// TIA Portal V20 export
VAR_GLOBAL   // PLC tag table "im"
   "i0.0" AT %I0.0 : Bool;
   "i0.1" AT %I0.1 : Bool;
   "i0.2" AT %I0.2 : Bool;
   "i0.3" AT %I0.3 : Bool;
   "i0.4" AT %I0.4 : Bool;
   "i0.5" AT %I0.5 : Bool;
   "i0.6" AT %I0.6 : Bool;
   "i0.7" AT %I0.7 : Bool;
   "i1.0" AT %I1.0 : Bool;
   "i1.1" AT %I1.1 : Bool;
   "i1.2" AT %I1.2 : Bool;
   "i1.3" AT %I1.3 : Bool;
   "i1.4" AT %I1.4 : Bool;
   "i1.5" AT %I1.5 : Bool;
   "i1.6" AT %I1.6 : Bool;
   "i1.7" AT %I1.7 : Bool;
   "i2.0" AT %I2.0 : Bool;
   "i2.1" AT %I2.1 : Bool;
   "i2.2" AT %I2.2 : Bool;
   "i2.3" AT %I2.3 : Bool;
   "i2.4" AT %I2.4 : Bool;
   "i2.5" AT %I2.5 : Bool;
   "i2.6" AT %I2.6 : Bool;
   "i2.7" AT %I2.7 : Bool;
   "i3.0" AT %I3.0 : Bool;
   "i3.1" AT %I3.1 : Bool;
   "i3.2" AT %I3.2 : Bool;
   "i3.3" AT %I3.3 : Bool;
   "i3.4" AT %I3.4 : Bool;
   "i3.5" AT %I3.5 : Bool;
   "i3.6" AT %I3.6 : Bool;
   "i3.7" AT %I3.7 : Bool;
   "i4.0" AT %I4.0 : Bool;
   "i4.1" AT %I4.1 : Bool;
   "i4.2" AT %I4.2 : Bool;
   "i4.3" AT %I4.3 : Bool;
   "i4.4" AT %I4.4 : Bool;
   "i4.5" AT %I4.5 : Bool;
   "i4.6" AT %I4.6 : Bool;
   "i4.7" AT %I4.7 : Bool;
   "i5.0" AT %I5.0 : Bool;
   "i5.1" AT %I5.1 : Bool;
   "i5.2" AT %I5.2 : Bool;
   "i5.3" AT %I5.3 : Bool;
   "i5.4" AT %I5.4 : Bool;
   "i5.5" AT %I5.5 : Bool;
   "i5.6" AT %I5.6 : Bool;
   "i5.7" AT %I5.7 : Bool;
   "i6.0" AT %I6.0 : Bool;
   "i6.1" AT %I6.1 : Bool;
   "i6.2" AT %I6.2 : Bool;
   "i6.3" AT %I6.3 : Bool;
   "i6.4" AT %I6.4 : Bool;
   "i6.5" AT %I6.5 : Bool;
   "i6.6" AT %I6.6 : Bool;
   "i6.7" AT %I6.7 : Bool;
   "i7.0" AT %I7.0 : Bool;
   "i7.1" AT %I7.1 : Bool;
   "i7.2" AT %I7.2 : Bool;
   "i7.3" AT %I7.3 : Bool;
   "i7.4" AT %I7.4 : Bool;
   "i7.5" AT %I7.5 : Bool;
   "i7.6" AT %I7.6 : Bool;
   "i7.7" AT %I7.7 : Bool;
   "q0.0" AT %Q0.0 : Bool;
   "q0.1" AT %Q0.1 : Bool;
   "q0.2" AT %Q0.2 : Bool;
   "q0.3" AT %Q0.3 : Bool;
   "q0.4" AT %Q0.4 : Bool;
   "q0.5" AT %Q0.5 : Bool;
   "q0.6" AT %Q0.6 : Bool;
   "q0.7" AT %Q0.7 : Bool;
   "q1.0" AT %Q1.0 : Bool;
   "q1.1" AT %Q1.1 : Bool;
   "q1.2" AT %Q1.2 : Bool;
   "q1.3" AT %Q1.3 : Bool;
   "q1.4" AT %Q1.4 : Bool;
   "q1.5" AT %Q1.5 : Bool;
   "q1.6" AT %Q1.6 : Bool;
   "q1.7" AT %Q1.7 : Bool;
   "q2.0" AT %Q2.0 : Bool;
   "q2.1" AT %Q2.1 : Bool;
   "q2.2" AT %Q2.2 : Bool;
   "q2.3" AT %Q2.3 : Bool;
   "q2.4" AT %Q2.4 : Bool;
   "q2.5" AT %Q2.5 : Bool;
   "q2.6" AT %Q2.6 : Bool;
   "q2.7" AT %Q2.7 : Bool;
   "q3.0" AT %Q3.0 : Bool;
   "q3.1" AT %Q3.1 : Bool;
   "q3.2" AT %Q3.2 : Bool;
   "q3.3" AT %Q3.3 : Bool;
   "q3.4" AT %Q3.4 : Bool;
   "q3.5" AT %Q3.5 : Bool;
   "q3.6" AT %Q3.6 : Bool;
   "q3.7" AT %Q3.7 : Bool;
   "q4.0" AT %Q4.0 : Bool;
   "q4.1" AT %Q4.1 : Bool;
   "q4.2" AT %Q4.2 : Bool;
   "q4.3" AT %Q4.3 : Bool;
   "q4.4" AT %Q4.4 : Bool;
   "q4.5" AT %Q4.5 : Bool;
   "q4.6" AT %Q4.6 : Bool;
   "q4.7" AT %Q4.7 : Bool;
   "q5.0" AT %Q5.0 : Bool;
   "q5.1" AT %Q5.1 : Bool;
   "q5.2" AT %Q5.2 : Bool;
   "q5.3" AT %Q5.3 : Bool;
   "q5.4" AT %Q5.4 : Bool;
   "q5.5" AT %Q5.5 : Bool;
   "q5.6" AT %Q5.6 : Bool;
   "q5.7" AT %Q5.7 : Bool;
   "q6.0" AT %Q6.0 : Bool;
   "q6.1" AT %Q6.1 : Bool;
   "q6.2" AT %Q6.2 : Bool;
   "q6.3" AT %Q6.3 : Bool;
   "q6.4" AT %Q6.4 : Bool;
   "q6.5" AT %Q6.5 : Bool;
   "q6.6" AT %Q6.6 : Bool;
   "q6.7" AT %Q6.7 : Bool;
   "q7.0" AT %Q7.0 : Bool;
   "q7.1" AT %Q7.1 : Bool;
   "q7.2" AT %Q7.2 : Bool;
   "q7.3" AT %Q7.3 : Bool;
   "q7.4" AT %Q7.4 : Bool;
   "q7.5" AT %Q7.5 : Bool;
   "q7.6" AT %Q7.6 : Bool;
   "q7.7" AT %Q7.7 : Bool;
END_VAR
